// TwinCAT 3 PLC project GetDeviceData
// Title: DeviceInfo
// Company: seehmatix
// Author: Matthias Seehauser
// ProjectVersion: 1.0.2.0
// ProgramVersion: 3.1.4026.12
// libraries:
//   Tc2_IoFunctions, 3.4.4.0 (Beckhoff Automation GmbH)
//   Tc2_Standard, * (Beckhoff Automation GmbH)
//   Tc2_System, * (Beckhoff Automation GmbH)
//   Tc2_Utilities, * (Beckhoff Automation GmbH)
//   Tc3_Module, * (Beckhoff Automation GmbH)
//   ZCore, 1.6.0.3 (Zeugwerk GmbH)
// project tree:
//   / DeviceInfo.TcPOU, DeviceInfoSteps.TcDUT, SlaveInfo.TcPOU, SlaveInfoSteps.TcDUT, Parameter.TcGVL

// ---- DeviceInfoSteps.TcDUT
{attribute 'qualified_only'}
TYPE DeviceInfoSteps :
(
	Begin,
  FetchDeviceTypes,
  ResetId1,
  GetDeviceNames,
  ResetId2,
  GetDeviceNetIds,
  End
);
END_TYPE

// ---- SlaveInfoSteps.TcDUT
{attribute 'qualified_only'}
TYPE SlaveInfoSteps :
(  
	Begin,
  FetchSlaveNames,
  End
);
END_TYPE

// ---- Parameter.TcGVL
{attribute 'qualified_only'}
VAR_GLOBAL CONSTANT
  MaxDevicesSearchCount : UINT := 200;
  MaxDeviceToBeFound : UINT := 10;
  MaxSlavesToBeFound : UINT := 200;
END_VAR

// ---- DeviceInfo.TcPOU
{attribute 'no_explicit_call'}
{attribute 'conditionalshow_all_locals'}
FUNCTION_BLOCK DeviceInfo EXTENDS ZCore.Object IMPLEMENTS ZCore.IUnmanagedObject
VAR_OUTPUT
  NameArray : ARRAY[0..Parameter.MaxDeviceToBeFound] OF ZCore.ZString;
  DeviceIdArray : ARRAY[0..Parameter.MaxDeviceToBeFound] OF UDINT;
  NetIdArray : ARRAY[0..Parameter.MaxDeviceToBeFound] OF Tc2_System.T_AmsNetID;
END_VAR
VAR
  _amsNetId : Tc2_System.T_AmsNetID;
  _ethercatMasterCount : UINT;
  _step : ZCore.Step(DeviceInfoSteps.Begin, DeviceInfoSteps.End);
END_VAR

/// The cyclic method should be run in any PLC-cycle. If the object has no work to do, we will simply
/// RETURN here. If an action has been started, this cyclic method takes care of all the work to do.
METHOD Cyclic
VAR_INST
  itIndex : UINT;
  ethercatMasters : UINT;

  getDeviceType : Tc2_IoFunctions.IOF_GetDeviceType;
  getDeviceName : Tc2_IoFunctions.IOF_GetDeviceName;
  getDeviceNetIds : Tc2_IoFunctions.IOF_GetDeviceNetId;
END_VAR
CASE _step.Index OF
  DeviceInfoSteps.Begin:
    IF Busy
    THEN
      ResetMem();
      _ethercatMasterCount := 0;
      _step.SetNext(DeviceInfoSteps.FetchDeviceTypes);
    END_IF
  
  DeviceInfoSteps.FetchDeviceTypes:
    IF _step.OnEntry()
    THEN
      getDeviceType(START:=FALSE);
      getDeviceType(START:=TRUE, NETID:=_amsNetId, DEVICEID:=ItIndex, TMOUT:=T#2S);
    END_IF
    
    getDeviceType(START:=FALSE);
    IF getDeviceType.ERR // no valid device found
    THEN
      IF ItIndex > Parameter.MaxDevicesSearchCount 
      THEN
        _step.SetNext(DeviceInfoSteps.ResetId1);
      ELSE
        _step.SetNext(DeviceInfoSteps.FetchDeviceTypes);
      END_IF
      
      itIndex := itIndex + 1;
    ELSIF NOT getDeviceType.BUSY
    THEN
      IF getDeviceType.IODeviceType = Tc2_IoFunctions.IODEVICETYPE_ETHERCAT
      THEN
        DeviceIdArray[_ethercatMasterCount] := itIndex;
        _ethercatMasterCount := _ethercatMasterCount + 1;
        itIndex := itIndex + 1;
        _step.SetNext(DeviceInfoSteps.ResetId1);
      END_IF
    END_IF

  DeviceInfoSteps.ResetId1:
    itIndex := 0;
    _step.SetNext(DeviceInfoSteps.GetDeviceNames);  
    
  DeviceInfoSteps.GetDeviceNames:
    IF _step.OnEntry()
    THEN
      getDeviceName(START:=FALSE);
      getDeviceName(START:=TRUE, NETID:=_amsNetId, DEVICEID:=DeviceIdArray[ItIndex], TMOUT:=T#2S);
    END_IF  
    
    getDeviceName();
    IF getDeviceName.ERR
    THEN
      Abort('Name could not be fetched!');
    ELSIF NOT getDeviceName.BUSY
    THEN
      NameArray[itIndex] := getDeviceName.DEVICENAME;
      itIndex := itIndex + 1;
      IF DeviceIdArray[itIndex] <> 0
      THEN
        _step.SetNext(DeviceInfoSteps.GetDeviceNames);
      ELSE
        _step.SetNext(DeviceInfoSteps.ResetId2);
      END_IF
    END_IF
    
  DeviceInfoSteps.ResetId2:
    itIndex := 0;
    _step.SetNext(DeviceInfoSteps.GetDeviceNetIds);  
    
  DeviceInfoSteps.GetDeviceNetIds:
    IF _step.OnEntry()
    THEN
      getDeviceNetIds(START:=FALSE);
      getDeviceNetIds(START:=TRUE, NETID:=_amsNetId, DEVICEID:=DeviceIdArray[itIndex], TMOUT:=T#2S);
    END_IF  
    
    getDeviceNetIds();
    IF getDeviceNetIds.ERR
    THEN
      Abort('Name could not be fetched!');
    ELSIF NOT getDeviceNetIds.BUSY
    THEN
      NetIdArray[itIndex] := getDeviceNetIds.DeviceNetId;
      itIndex := itIndex + 1;
      IF DeviceIdArray[itIndex] = 0
      THEN
        SetBusy(FALSE);
        _step.SetNext(DeviceInfoSteps.End);
      END_IF
    END_IF      
  
  DeviceInfoSteps.End:
    RETURN;
    
END_CASE
END_METHOD

/// Returns the actual found Ethercat Master count -> Needed to iterate through the VAR_INPUT Arrays of AMSNet-IDs and
/// Ethercat Master Device names.
PROPERTY EthercatMasterCount : UINT
GET
EthercatMasterCount := _ethercatMasterCount;
END_GET
END_PROPERTY

/// Sets the object to Idle-State becuse no booting phase is needed here!
METHOD FB_init : BOOL
VAR_INPUT
	bInitRetains : BOOL; // if TRUE, the retain variables are initialized (warm start / cold start)
	bInCopyCode : BOOL;  // if TRUE, the instance afterwards gets moved into the copy code (online change)
END_VAR
SetIdle();
END_METHOD

/// Starts reading of all available Ethercat-Master Device names
/// Just wait until Busy property of this object returns FALSE -> then fetch all Ethercat Master names from
/// the Array in VAR_INPUT of this object
METHOD ReadDeviceNamesAsync
VAR_INPUT
  amsNetId : Tc2_System.T_AmsNetID; //< AMS-Netid of the IPC on which the device names should be fetched
END_VAR
SetBusy(TRUE);
_amsNetId := amsNetId;
_step.SetNext(DeviceInfoSteps.Begin);
END_METHOD

METHOD PRIVATE ResetMem
VAR
  count : UINT;
END_VAR
FOR count:=0 TO Parameter.MaxDeviceToBeFound BY 1 DO
  NameArray[count] := '';
  DeviceIdArray[count] := 0;
  NetIdArray[count] := '';
END_FOR
END_METHOD

END_FUNCTION_BLOCK

// ---- SlaveInfo.TcPOU
{attribute 'no_explicit_call'}
{attribute 'conditionalshow_all_locals'}
FUNCTION_BLOCK SlaveInfo EXTENDS ZCore.Object IMPLEMENTS ZCore.IUnmanagedObject
VAR_OUTPUT
  NameArray : ARRAY[0..Parameter.MaxSlavesToBeFound] OF ZCore.ZString;
  PortArray : ARRAY[0..Parameter.MaxSlavesToBeFound] OF UINT;
END_VAR
VAR
  _amsNetId : Tc2_System.T_AmsNetID;
  _deviceId : UDINT;
  _ethercatSlavesCount : UINT;
  _step : ZCore.Step(SlaveInfoSteps.Begin, SlaveInfoSteps.End);
END_VAR

METHOD Cyclic
VAR_INST
  getBoxNameByAddr : Tc2_IoFunctions.IOF_GetBoxNameByAddr;
  boxAddrIterator : UINT;
END_VAR
VAR CONSTANT
  FirstSlaveAddr : UINT := 1001;
END_VAR
CASE _step.Index OF
  SlaveInfoSteps.Begin:
    IF Busy
    THEN
      ResetMem();
      _ethercatSlavesCount := 0;
      boxAddrIterator := 1001;
      _step.SetNext(DeviceInfoSteps.FetchDeviceTypes);
    END_IF
  
  SlaveInfoSteps.FetchSlaveNames:
    IF _step.OnEntry()
    THEN
      getBoxNameByAddr(START:=FALSE);
      getBoxNameByAddr(START:=TRUE, NETID:=_amsNetId, DEVICEID:=_deviceId, BOXADDR:=boxAddrIterator, TMOUT:=T#2S);
    END_IF
    
    getBoxNameByAddr(START:=FALSE);
    IF getBoxNameByAddr.ERR // no valid device found
    THEN
      SetBusy(FALSE);
      _step.SetNext(DeviceInfoSteps.End);
    ELSIF NOT getBoxNameByAddr.BUSY
    THEN
      // first slave starts on address 1001
      IF boxAddrIterator > (Parameter.MaxSlavesToBeFound + FirstSlaveAddr)
      THEN
        Abort('MaxSlavesToBeFound Parameter reached! Consider raising MaxSlavesToBeFound Parameter of library...');
        _step.SetNext(SlaveInfoSteps.End);
      ELSE
        NameArray[boxAddrIterator-FirstSlaveAddr] := getBoxNameByAddr.BOXNAME;
        PortArray[boxAddrIterator-FirstSlaveAddr] := boxAddrIterator;
        boxAddrIterator := boxAddrIterator + 1;
        _step.RepeatStep();
			END_IF
    END_IF
  
  SlaveInfoSteps.End:
    RETURN;
    
END_CASE
END_METHOD

PROPERTY EthercatSlavesCount : UINT
GET
END_GET
END_PROPERTY

METHOD FB_init : BOOL
VAR_INPUT
	bInitRetains : BOOL; // if TRUE, the retain variables are initialized (warm start / cold start)
	bInCopyCode : BOOL;  // if TRUE, the instance afterwards gets moved into the copy code (online change)
END_VAR
SetIdle();
END_METHOD

/// Starts reading of all available Ethercat-Slave Box names for a given DeviceId/Ethercat-Master
/// Just wait until Busy property of this object returns FALSE (or the object is DONE=TRUE) -> then fetch all Ethercat Slave names from
/// the Array in VAR_INPUT of this object
METHOD ReadSlaveNamesAsync
VAR_INPUT
  amsNetId : Tc2_System.T_AmsNetID; //< AMS-Netid of the IPC on which the Ethercat-Slave names should be fetched from a given Master DeviceID
  deviceId : UDINT; //< DeviceID of a Ethercat-Master from which all Ethercat-Slave names should be fetched
END_VAR
SetBusy(TRUE);
_deviceId := deviceId;
_amsNetId := amsNetId;
_step.SetNext(SlaveInfoSteps.Begin);
END_METHOD

METHOD PRIVATE ResetMem
VAR
  count : UINT;
END_VAR
FOR count:=0 TO Parameter.MaxSlavesToBeFound BY 1 DO
  NameArray[count] := '';
  PortArray[count] := 0;
END_FOR
END_METHOD

END_FUNCTION_BLOCK
